(* IEC 61131-3 sources: CodesysTest/export/SX_1195.dev/Plc Logic/Application, 9 files *)

(* ---- AxisData.gvl.st ---- *)
(*#-#-#-#-#-#-#-#-#-#---Declaration---#-#-#-#-#-#-#-#-#-#-#-#-#*)

{attribute 'qualified_only'}
//{attribute 'global_init_slot' := '49994'}
VAR_GLOBAL PERSISTENT

	(* Jaw *)
	jawJogMotionProfile : sctMotionProfile := (
		acceleration := 200,
		deceleration := 200,
		velocity := 2,
		minPosition := 0,
		maxPosition := 5.5,
		current := 30.0
	);
	jawConfig : sctAxisConfig := (
		stepsPerInch := 2410,
		rotationsPerInch := 0.241,
		zeroOffset := 0,
		defaultCurrent := 100.0
	);

	jawOpenMotionProfile : sctMotionProfile := (
		acceleration := 100,
		deceleration := 100,
		velocity := 30.0,
		current := 100.0,
		position := 5.5
	);

	jawCloseMotionProfile : sctMotionProfile := (
		acceleration := 100,
		deceleration := 100,
		velocity := 30.0,
		current := 100.0,
		position := -0.5
	);

	jawPushMotionProfile : sctMotionProfile := (
		acceleration := 100,
		deceleration := 100,
		velocity := 4,
		current := 100.0,
		position := -1
	);

	(* Load Plate *)

	loadPlateConfig : sctAxisConfig := (
		stepsPerInch := 9310,
		rotationsPerInch := 0.931,
		zeroOffset := 0.0
	);

	loadPlateRaiseMotionProfile : sctMotionProfile := (
		acceleration := 300000.0,
		deceleration := 300000.0,
		velocity := 10.0,
		current := 100.0
	);

	loadPlateLowerMotionProfile : sctMotionProfile := (
		acceleration := 300000.0,
		deceleration := 300000.0,
		velocity := 10000.0,
		current := 100.0
	);

	(* IBD *)

	IBDConfig : sctAxisConfig := (
		stepsPerInch := 12500,
		rotationsPerInch := 1.25,
		zeroOffset := 2.0
	);

	IBDJogMotionProfile : sctMotionProfile := (
		acceleration := 0,
		deceleration := 0,
		velocity := 0,
	 	minPosition := 0,
		maxPosition := 0
	);

	IBDOpenMotionProfile : sctMotionProfile := (
		acceleration := 300000.0,
 		deceleration := 300000.0,
		velocity := 10000.0,
		current := 100.0
	);

	IBDCloseMotionProfile : sctMotionProfile := (
		acceleration := 300000.0,
 		deceleration := 300000.0,
		velocity := 10.0,
		current := 50.0
	);

	(* Film Feed *)

	FilmFeedConfig : sctAxisConfig := (
		stepsPerInch := 4900,
		rotationsPerInch := 0.490,
		zeroOffset := 2.0,
		defaultCurrent := 100.0
	);

	FilmFeedJogMotionProfile : sctMotionProfile := (
		acceleration := 200,
		deceleration := 200,
		velocity := 2,
	 	minPosition := -20,
		maxPosition := 20,
		position := 20,
		current := 100
	);

	FilmFeedForwardMotionProfile : sctMotionProfile := (
		acceleration := 75,
 		deceleration := 100,
		velocity := 60,
		position := 17.5,
		current := 100.0
	);

	FilmFeedReverseMotionProfile : sctMotionProfile := (
		acceleration := 50,
 		deceleration := 50,
		velocity := 12,
		position := -1,
		current := 100.0
	);

	FilmFeedPrintMotionProfile : sctMotionProfile := (
		acceleration := 100,
 		deceleration := 100,
		velocity := 12,
		position := -1,
		current := 100.0
	);

	FilmFeedPrintOffsetMotionProfile : sctMotionProfile := (
		acceleration := 75,
 		deceleration := 100,
		velocity := 12,
		position := -1,
		current := 100.0
	);

END_VAR

VAR_GLOBAL
	jaw : sctAxisData := (
		config := jawConfig,
		jogType := eDiscreteMotionType.Absolute
	);

	FilmFeed : sctAxisData := (
		config := FilmFeedConfig,
		jogType := eDiscreteMotionType.Relative
	);

	IBD : sctAxisData := (
		config := IBDConfig,
		jogType := eDiscreteMotionType.Absolute
	);

	loadPlate : sctAxisData := (
		config := loadPlateConfig
	);
END_VAR

(* ---- Counters.gvl.st ---- *)
(*#-#-#-#-#-#-#-#-#-#---Declaration---#-#-#-#-#-#-#-#-#-#-#-#-#*)

{attribute 'qualified_only'}
VAR_GLOBAL
	jawCycleTestCount : FB_MachineCounter(name := 'Jaw Cycle Test Counter');
	baggerCycles : FB_MachineCounter(name := 'Bagger Cycle Counter');
	pressureBarCycles : FB_MachineCounter(name := 'Pressure Bar Cycle Counter');

	(*Counters*)

	//passthroughChanges : FB_MachineCounter(name := 'Passthrough Changes Counter');
	//loadPlateCycles : FB_MachineCounter(name := 'Load Plate Cycle Counter');
	//printerCycles : FB_MachineCounter(name := 'Printer Cycle Counter');
	//motorizedSealFlattenerCycles : FB_MachineCounter(name := 'Motorized Seal Flattener Cycles');
	//bagOpenRetryTotal : FB_MachineCounter(name := 'Bag Open Retry Totals');
END_VAR

(* ---- GlobalData.gvl.st ---- *)
(*#-#-#-#-#-#-#-#-#-#---Declaration---#-#-#-#-#-#-#-#-#-#-#-#-#*)

{attribute 'qualified_only'}
{attribute 'global_init_slot' := '49994'}
VAR_GLOBAL
	SystemLog : FB_InternalLogger;
END_VAR

VAR_GLOBAL CONSTANT
	MAX_LOGGED_ITEMS : UINT := 500;	// Max items to be logged
	STEPS_PER_INCH_IBD : DINT := 1250;
	STEPS_PER_INCH_JAW : DINT := 1250;
	STEPS_PER_INCH_LOAD_PLATE : DINT := 931;
	STEPS_PER_INCH_FILM : DINT := 1000;
	SERIAL_BUFFER_SIZE : BYTE := 50;
	SEAL_TO_PHOTOEYE_DISTANCE : REAL := 3.25;
END_VAR

(* ---- IO.gvl.st ---- *)
(*#-#-#-#-#-#-#-#-#-#---Declaration---#-#-#-#-#-#-#-#-#-#-#-#-#*)

{attribute 'qualified_only'}
{attribute 'global_init_slot' := '50010'}
VAR_GLOBAL
	iptJawNotObstructed : FB_PhysicalDigitalInput(name := 'Jaw Not Obstructed') := (in := iJawNotObstructed);
	iptPrinterDataReady : FB_PhysicalDigitalInput(name := 'Printer Data Ready') := (in := iPrinterDataReady);
	iptPrinterBusy : FB_PhysicalDigitalInput(name := 'Printer Busy') := (in := iPrinterBusy);
	iptBagEdgePhotoeye : FB_PhysicalDigitalInput(name := 'Bag Edge Photoeye') := (in := iBagEdgePhotoeye);
	iptCycleStart : FB_PhysicalDigitalInput(name := 'Cycle Start') := (in := iCycleStart);
	iptPrintHeadLowered : FB_PhysicalDigitalInput(name := 'Printhead Lowered') := (in := iPrintHeadLowered);
	iptJawClosed : FB_PhysicalDigitalInput(name := 'Jaw Closed') := (in := iJawClosed);
	iptJawNearClosed : FB_PhysicalDigitalInput(name := 'Jaw Near Closed') := (in := iJawNearClosed);
	iptBarcodeOK : FB_PhysicalDigitalInput(name := 'Barcode OK') := (in := iBarcodeOK);
	iptBarcodeNG : FB_PhysicalDigitalInput(name := 'Barcode NG') := (in := iBarcodeNG);
	iptLightCurtain : FB_PhysicalDigitalInput(name := 'Light Curtain Clear') := (in := iLightCurtain);
	iptFillerTrigger : FB_PhysicalDigitalInput(name := 'Filler Trigger') := (in := iFillerTrigger);
	iptLHPalmButton : FB_PhysicalDigitalInput(name := 'LH Palm Button') := (in := iLHPalmButton);
	iptRHPalmButton : FB_PhysicalDigitalInput(name := 'RH Palm Button') := (in := iRHPalmButton);
	iptTopCoverClosed : FB_PhysicalDigitalInput(name := 'Top Cover Closed') := (in := iTopCoverClosed);
	iptPrinterRibbonEncoder : FB_PhysicalDigitalInput(name := 'Top Cover Closed') := (in := iPrinterRibbonEncoder);

	outSealWire : FB_PhysicalDigitalOutput(name := 'Seal Wire Output') := (refOutput := oSealWire);
	outLowerPrintHead : FB_PhysicalDigitalOutput(name := 'Lower Printhead') := (refOutput := oLowerPrintHead);
	outRequestPrint : FB_PhysicalDigitalOutput(name := 'Request Print') := (refOutput := oRequestPrint);
	outPrinterRibbonUnwind : FB_PhysicalDigitalOutput(name := 'Ribbon Unwind') := (refOutput := oPrinterRibbonUnwind);
	outTriggerBCV : FB_PhysicalDigitalOutput(name := 'Trigger BCV') := (refOutput := oTriggerBCV);
	outTeachPhotoeye : FB_PhysicalDigitalOutput(name := 'Teach Photoeye') := (refOutput := oTeachPhotoeye);
	outRedStackLight : FB_PhysicalDigitalOutput(name := 'Red Stack Light') := (refOutput := oRedStackLight);
	outGreenStackLight : FB_PhysicalDigitalOutput(name := 'Green Stack Light') := (refOutput := oGreenStackLight);
	outReadyForFiller : FB_PhysicalDigitalOutput(name := 'Ready for Filler') := (refOutput := oReadyForFiller);
	outPalmButton0 : FB_PhysicalDigitalOutput(name := 'Palm Button 0') := (refOutput := oPalmButton0);
	outPalmButton1 : FB_PhysicalDigitalOutput(name := 'Palm Button 1') := (refOutput := oPalmButton1);
END_VAR

(* ---- IO_Mapping.gvl.st ---- *)
(*#-#-#-#-#-#-#-#-#-#---Declaration---#-#-#-#-#-#-#-#-#-#-#-#-#*)

VAR_GLOBAL
	mainIOamax4830Input: ARRAY[0..15] OF universalIOObject;
	mainIOamax4830Output: ARRAY[0..15] OF universalIOObject;
	oSealWire: REFERENCE TO BOOL;
	oLowerPrinthead: Reference to BOOL;
	oRequestPrint: Reference to BOOL;
	oPrinterRibbonUnwind: Reference to BOOL;
	oTriggerBCV: Reference to BOOL;
	oFansEnable: Reference to BOOL;
	oPalmButton0: Reference to BOOL;
	oPalmButton1: Reference to BOOL;
	oPbarClampMotorStart: Reference to BOOL;
	oPbarClampMotorReverse: Reference to BOOL;
	oPbarClampMotorAlarmReset: Reference to BOOL;
	iPrinterServiceRequired: Reference to BOOL;
	iPrinterDataReady: Reference to BOOL;
	iPrinterBusy: Reference to BOOL;
	iBagEdgePhotoeye: Reference to BOOL;
	iCycleStart: Reference to BOOL;
	iPbarClampMotorAlarm: Reference to BOOL;
	iClampHomeSensor: Reference to BOOL;
	iJawNotObstructed: Reference to BOOL;
	iBarcodeOK: Reference to BOOL;
	iBarcodeNG: Reference to BOOL;
	iLightCurtainClear: Reference to BOOL;
	iTopCoverClosed: Reference to BOOL;
	iPrinterRibbonEncoder: REFERENCE TO BOOL;
END_VAR

(* ---- PersistentVars.gvl.st ---- *)
(*#-#-#-#-#-#-#-#-#-#---Declaration---#-#-#-#-#-#-#-#-#-#-#-#-#*)

VAR_GLOBAL RETAIN PERSISTENT
	// Generated instance path of persistent variable
	PLC_PRG_1.baggerCM.dualMotorPassthrough.factoryHomeJaw: BOOL;
	// Generated instance path of persistent variable
	HMIData.bagsMade: UDINT;
	// Generated instance path of persistent variable
	HMIData.batchEnable: BOOL;
	// Generated instance path of persistent variable
	HMIData.batchSetting: UDINT := UDINT#10;
	// Generated instance path of persistent variable
	HMIData.batchCount: UDINT;
	// Generated instance path of persistent variable
	HMIData.headCycleCount: UDINT;
	// Generated instance path of persistent variable
	HMIData.pressureBarOpenDelay: REAL;
	// Generated instance path of persistent variable
	HMIData.pressureBarCloseDelay: REAL;
	// Generated instance path of persistent variable
	HMIData.passthroughSetting: REAL := REAL#5.5;
	// Generated instance path of persistent variable
	HMIData.sealBarDwell: REAL := REAL#0.2;
	// Generated instance path of persistent variable
	HMIData.sealBarCool: REAL := REAL#0.4;
	// Generated instance path of persistent variable
	HMIData.bagSkirtLength: REAL := 2.0;
	// Generated instance path of persistent variable
	HMIData.bagLength: REAL := REAL#17.62;
	// Generated instance path of persistent variable
	HMIData.bagWidth: REAL := 11.0;
	// Generated instance path of persistent variable
	HMIData.bagThickness: REAL := REAL#2.5;
	// Generated instance path of persistent variable
	HMIData.bagForwardSpeed: UDINT := UDINT#40;
	// Generated instance path of persistent variable
	HMIData.bagReverseSpeed: UDINT := UDINT#8;
	// Generated instance path of persistent variable
	HMIData.printSpeed: UINT := UINT#6;
	// Generated instance path of persistent variable
	HMIData.printLength: REAL := REAL#1.25;
	// Generated instance path of persistent variable
	HMIData.printOffset: REAL := REAL#9;
	// Generated instance path of persistent variable
	HMIData.fillerCountSetting: UDINT;
	// Generated instance path of persistent variable
	HMIData.fillerCurrentCount: UDINT;
	// Generated instance path of persistent variable
	HMIData.fillerDropTime: REAL;
	// Generated instance path of persistent variable
	HMIData.loadPlateDelay: REAL;
	// Generated instance path of persistent variable
	HMIData.loadPlateDwell: REAL := REAL#0.1;
	// Generated instance path of persistent variable
	HMIData.IBDInUse: BOOL;
	// Generated instance path of persistent variable
	HMIData.IBDInstalled: BOOL := FALSE;
	// Generated instance path of persistent variable
	HMIData.jawCloseDelay: REAL := REAL#0.1;
	// Generated instance path of persistent variable
	HMIData.jawClosePositionSetting: REAL := REAL#-0.45;
	// Generated instance path of persistent variable
	HMIData.lastCycleTime: REAL;
	// Generated instance path of persistent variable
	HMIData.bagDropClearanceDwell: REAL := REAL#0.5;
	// Generated instance path of persistent variable
	HMIData.averageCycleTime: REAL;
	// Generated instance path of persistent variable
	HMIData.currentJobID: INT;
	// Generated instance path of persistent variable
	HMIData.separateBeforeSeal: BOOL := TRUE;
	// Generated instance path of persistent variable
	HMIData.partsCounterEnable: BOOL;
	// Generated instance path of persistent variable
	HMIData.partsCounterCount: UDINT;
	// Generated instance path of persistent variable
	HMIData.partsCounterSetting: UDINT;
	// Generated instance path of persistent variable
	HMIData.consecutiveBagsEnable: BOOL;
	// Generated instance path of persistent variable
	HMIData.consecutiveBagsCount: UDINT;
	// Generated instance path of persistent variable
	HMIData.consecutiveBagsSetting: UDINT;
	// Generated instance path of persistent variable
	HMIData.printerInstalled: BOOL := FALSE;
	// Generated instance path of persistent variable
	HMIData.printerInUse: BOOL := FALSE;
	// Generated instance path of persistent variable
	HMIData.printerCancelRequest: BOOL;
	// Generated instance path of persistent variable
	HMIData.barcodeVerifierInstalled: BOOL := FALSE;
	// Generated instance path of persistent variable
	HMIData.barcodeGoodReadCount: UDINT;
	// Generated instance path of persistent variable
	HMIData.barcodeBadReadCount: UDINT;
	// Generated instance path of persistent variable
	HMIData.barcodeBadReadFaultSetting: UDINT := UDINT#1;
	// Generated instance path of persistent variable
	HMIData.barcodeStartPosition: REAL := REAL#4.5;
	// Generated instance path of persistent variable
	HMIData.barcodeScanDistance: REAL := REAL#0.1;
	// Generated instance path of persistent variable
	HMIData.barcodeVerifierInUse: BOOL;
	// Generated instance path of persistent variable
	HMIData.loadPlateInstalled: BOOL := FALSE;
	// Generated instance path of persistent variable
	HMIData.loadPlateLoweredPositionSetting: REAL := 0.0;
	// Generated instance path of persistent variable
	HMIData.loadPlateRaisedPositionSetting: REAL := 1.0;
	// Generated instance path of persistent variable
	HMIData.loadPlateInUse: BOOL;
	// Generated instance path of persistent variable
	HMIData.fillerEnable: BOOL;
	// Generated instance path of persistent variable
	HMIData.autoModeEnable: BOOL;
	// Generated instance path of persistent variable
	HMIData.autoModeDwell: REAL;
	// Generated instance path of persistent variable
	HMIData.dryCycleEnable: BOOL;
	// Generated instance path of persistent variable
	HMIData.standbyTimeSetting: REAL := REAL#5;
	// Generated instance path of persistent variable
	HMIData.jawClampTime: REAL := REAL#1;
	// Generated instance path of persistent variable
	HMIData.jawClampReverseTime: REAL := REAL#1;
	// Generated instance path of persistent variable
	HMIData.jawClampInterval: REAL := REAL#2;
	// Generated instance path of persistent variable
	HMIData.jawEnableClamping: BOOL;
	// Generated instance path of persistent variable
	HMIData.jawCycleTestCycles: DINT;
	// Generated instance path of persistent variable
	HMIData.jawClampTestCycles: DINT;
	// Generated instance path of persistent variable
	HMIData.filmFeedTestCycles: DINT;
	// Generated instance path of persistent variable
	HMIData.jawEnableMotion: BOOL;
	// Generated instance path of persistent variable
	HMIData.filmEnableMotion: BOOL;
	// Generated instance path of persistent variable
	HMIData.printer300DPI: BOOL;
	// Generated instance path of persistent variable
	AxisData.jawJogMotionProfile: sctMotionProfile := STRUCT(acceleration := 200.0, deceleration := 200.0, velocity := 2.0, minPosition := REAL#0.0, maxPosition := 5.5, current := REAL#30);
	// Generated instance path of persistent variable
	AxisData.jawConfig: sctAxisConfig := STRUCT(stepsPerInch := 2410.0, rotationsPerInch := REAL#0.241, zeroOffset := 0.0, defaultCurrent := REAL#100);
	// Generated instance path of persistent variable
	AxisData.jawOpenMotionProfile: sctMotionProfile := STRUCT(acceleration := 100.0, deceleration := 100.0, velocity := REAL#30, current := REAL#100, position := REAL#5.5);
	// Generated instance path of persistent variable
	AxisData.jawCloseMotionProfile: sctMotionProfile := STRUCT(acceleration := 100.0, deceleration := 100.0, velocity := REAL#30, current := REAL#100, position := REAL#-0.5);
	// Generated instance path of persistent variable
	AxisData.jawPushMotionProfile: sctMotionProfile := STRUCT(acceleration := 100.0, deceleration := 100.0, velocity := 4.0, current := REAL#100, position := -1.0);
	// Generated instance path of persistent variable
	AxisData.loadPlateConfig: sctAxisConfig := STRUCT(stepsPerInch := 9310.0, rotationsPerInch := REAL#0.931, zeroOffset := REAL#0);
	// Generated instance path of persistent variable
	AxisData.loadPlateRaiseMotionProfile: sctMotionProfile := STRUCT(acceleration := REAL#300000, deceleration := REAL#300000, velocity := REAL#10, current := REAL#100);
	// Generated instance path of persistent variable
	AxisData.loadPlateLowerMotionProfile: sctMotionProfile := STRUCT(acceleration := REAL#300000, deceleration := REAL#300000, velocity := REAL#10000, current := REAL#100);
	// Generated instance path of persistent variable
	AxisData.IBDConfig: sctAxisConfig := STRUCT(stepsPerInch := 12500.0, rotationsPerInch := REAL#1.25, zeroOffset := REAL#2);
	// Generated instance path of persistent variable
	AxisData.IBDJogMotionProfile: sctMotionProfile := STRUCT(acceleration := 0.0, deceleration := 0.0, velocity := 0.0, minPosition := 0.0, maxPosition := 0.0);
	// Generated instance path of persistent variable
	AxisData.IBDOpenMotionProfile: sctMotionProfile := STRUCT(acceleration := REAL#300000, deceleration := REAL#300000, velocity := REAL#10000, current := REAL#100);
	// Generated instance path of persistent variable
	AxisData.IBDCloseMotionProfile: sctMotionProfile := STRUCT(acceleration := REAL#300000, deceleration := REAL#300000, velocity := REAL#10, current := REAL#50);
	// Generated instance path of persistent variable
	AxisData.FilmFeedConfig: sctAxisConfig := STRUCT(stepsPerInch := 4900.0, rotationsPerInch := REAL#0.49, zeroOffset := REAL#2, defaultCurrent := REAL#100);
	// Generated instance path of persistent variable
	AxisData.FilmFeedJogMotionProfile: sctMotionProfile := STRUCT(acceleration := 10.0, deceleration := 200.0, velocity := 100.0, minPosition := -20.0, maxPosition := 20.0, position := 20.0, current := 100.0);
	// Generated instance path of persistent variable
	AxisData.FilmFeedForwardMotionProfile: sctMotionProfile := STRUCT(acceleration := 75.0, deceleration := 100.0, velocity := 60.0, position := REAL#17.5, current := REAL#100);
	// Generated instance path of persistent variable
	AxisData.FilmFeedReverseMotionProfile: sctMotionProfile := STRUCT(acceleration := 50.0, deceleration := 50.0, velocity := 12.0, position := -1.0, current := REAL#100);
	// Generated instance path of persistent variable
	AxisData.FilmFeedPrintMotionProfile: sctMotionProfile := STRUCT(acceleration := 100.0, deceleration := 100.0, velocity := 12.0, position := -1.0, current := REAL#100);
	// Generated instance path of persistent variable
	AxisData.FilmFeedPrintOffsetMotionProfile: sctMotionProfile := STRUCT(acceleration := 75.0, deceleration := 100.0, velocity := 12.0, position := -1.0, current := REAL#100);
END_VAR

(* ---- IO_Map.pou.st ---- *)
(*#-#-#-#-#-#-#-#-#-#---Declaration---#-#-#-#-#-#-#-#-#-#-#-#-#*)

PROGRAM IO_Map
VAR
END_VAR
(*#-#-#-#-#-#-#-#-#-#---Implementation---#-#-#-#-#-#-#-#-#-#-#-#-#*)

//Output Configuration

oSealWire REF= IO_Mapping.mainIOamax4830Output[0].discreteSignal;
oLowerPrinthead REF= IO_Mapping.mainIOamax4830Output[1].discreteSignal;
oRequestPrint REF=IO_Mapping.mainIOamax4830Output[2].discreteSignal;
oPrinterRibbonUnwind REF=IO_Mapping.mainIOamax4830Output[3].discreteSignal;
oTriggerBCV REF=IO_Mapping.mainIOamax4830Output[4].discreteSignal;
//IO_Mapping.mainIOamax4830Output[5].discreteSignal;
oFansEnable REF=IO_Mapping.mainIOamax4830Output[6].discreteSignal;
//IO_Mapping.mainIOamax4830Output[7].discreteSignal;
//IO_Mapping.mainIOamax4830Output[8].discreteSignal;
oPalmButton0 REF=IO_Mapping.mainIOamax4830Output[9].discreteSignal;
oPalmButton1 REF=IO_Mapping.mainIOamax4830Output[10].discreteSignal;
oPbarClampMotorStart REF=IO_Mapping.mainIOamax4830Output[11].discreteSignal;
oPbarClampMotorReverse REF=IO_Mapping.mainIOamax4830Output[12].discreteSignal;
oPbarClampMotorAlarmReset REF=IO_Mapping.mainIOamax4830Output[13].discreteSignal;
//IO_Mapping.mainIOamax4830Output[14].discreteSignal;
//IO_Mapping.mainIOamax4830Output[15].discreteSignal;

IO_Mapping.mainIOamax4830Output[0].signalCommonName := 'O0\0: Seal Wire';
IO_Mapping.mainIOamax4830Output[1].signalCommonName := 'O0\1: Lower Print Head';
IO_Mapping.mainIOamax4830Output[2].signalCommonName := 'O0\2: Request Print';
IO_Mapping.mainIOamax4830Output[3].signalCommonName := 'O0\3: Printer Ribbon Unwind';
IO_Mapping.mainIOamax4830Output[4].signalCommonName := 'O0\4: Trigger Barcode Verification';
IO_Mapping.mainIOamax4830Output[5].signalCommonName := 'O0\5: Spare';
IO_Mapping.mainIOamax4830Output[6].signalCommonName := 'O0\6: Fans Enable';
IO_Mapping.mainIOamax4830Output[7].signalCommonName := 'O0\7: Spare';
IO_Mapping.mainIOamax4830Output[8].signalCommonName := 'O0\8: Spare';
IO_Mapping.mainIOamax4830Output[9].signalCommonName := 'O0\9: Palm Button 0';
IO_Mapping.mainIOamax4830Output[10].signalCommonName := 'O0\10: Palm Button 1';
IO_Mapping.mainIOamax4830Output[11].signalCommonName := 'O0\11: Pbar Clamp Motor Start';
IO_Mapping.mainIOamax4830Output[12].signalCommonName := 'O0\12: Pbar Clamp Motor Reverse';
IO_Mapping.mainIOamax4830Output[13].signalCommonName := 'O0\13: Pbar Clamp Motor Alarm Reset';
IO_Mapping.mainIOamax4830Output[14].signalCommonName := 'O0\14: Spare';
IO_Mapping.mainIOamax4830Output[15].signalCommonName := 'O0\15: Spare';

//Input Configuration

iPrinterServiceRequired REF= IO_Mapping.mainIOamax4830Input[0].discreteSignal;
iPrinterDataReady REF= IO_Mapping.mainIOamax4830Input[1].discreteSignal;
iPrinterBusy REF= IO_Mapping.mainIOamax4830Input[2].discreteSignal;
iBagEdgePhotoeye REF= IO_Mapping.mainIOamax4830Input[3].discreteSignal;
iCycleStart REF= IO_Mapping.mainIOamax4830Input[4].discreteSignal;
iPbarClampMotorAlarm REF= IO_Mapping.mainIOamax4830Input[5].discreteSignal;
iClampHomeSensor REF= IO_Mapping.mainIOamax4830Input[6].discreteSignal;
iJawNotObstructed REF= IO_Mapping.mainIOamax4830Input[7].discreteSignal;
iBarcodeOK REF= IO_Mapping.mainIOamax4830Input[8].discreteSignal;
iBarcodeNG REF= IO_Mapping.mainIOamax4830Input[9].discreteSignal;
iLightCurtainClear REF= IO_Mapping.mainIOamax4830Input[10].discreteSignal;
//IO_Mapping.mainIOamax4830Input[11].discreteSignal;
//IO_Mapping.mainIOamax4830Input[12].discreteSignal;
//IO_Mapping.mainIOamax4830Input[13].discreteSignal;
iTopCoverClosed REF= IO_Mapping.mainIOamax4830Input[14].discreteSignal;
iPrinterRibbonEncoder REF= IO_Mapping.mainIOamax4830Input[15].discreteSignal;

IO_Mapping.mainIOamax4830Input[0].signalCommonName := 'I0\0: Printer Service Required';
IO_Mapping.mainIOamax4830Input[1].signalCommonName := 'I0\1: Printer Data Ready';
IO_Mapping.mainIOamax4830Input[2].signalCommonName := 'I0\2: Printer Busy';
IO_Mapping.mainIOamax4830Input[3].signalCommonName := 'I0\3: Bag Edge Detect Photoeye';
IO_Mapping.mainIOamax4830Input[4].signalCommonName := 'I0\4: Cycle Start';
IO_Mapping.mainIOamax4830Input[5].signalCommonName := 'I0\5: Pbar Clamp Motor Alarm';
IO_Mapping.mainIOamax4830Input[6].signalCommonName := 'I0\6: Clamp Home Sensor';
IO_Mapping.mainIOamax4830Input[7].signalCommonName := 'I0\7: Jaw Not Obstructed';
IO_Mapping.mainIOamax4830Input[8].signalCommonName := 'I0\8: Bracode OK';
IO_Mapping.mainIOamax4830Input[9].signalCommonName := 'I0\9: Bracode NG';
IO_Mapping.mainIOamax4830Input[10].signalCommonName := 'I0\10: Light Curtain Clear';
IO_Mapping.mainIOamax4830Input[11].signalCommonName := 'I0\11: Spare';
IO_Mapping.mainIOamax4830Input[12].signalCommonName := 'I0\12: Spare';
IO_Mapping.mainIOamax4830Input[13].signalCommonName := 'I0\13: Spare';
IO_Mapping.mainIOamax4830Input[14].signalCommonName := 'I0\14: Top Cover Closed';
IO_Mapping.mainIOamax4830Input[15].signalCommonName := 'I0\15: Printer Ribbon Encoder';

(* ---- PLC_PRG.pou.st ---- *)
(*#-#-#-#-#-#-#-#-#-#---Declaration---#-#-#-#-#-#-#-#-#-#-#-#-#*)

PROGRAM PLC_PRG
VAR
	firstScanDone: BOOL;
	cycleStartONS : FB_ONS;
	powerUpFrontJawMotor : MC_Power;
	powerUpRearJawMotor : MC_Power;
	powerUpBothJawMotors : MC_Power;
	powerUpLoadPlateMotor : MC_Power;
	powerUpBagDeliveryMotor : MC_Power;
	powerUpIBDMotor : MC_Power;
	UN00_SXMachine : FB_UN00_SharpMachine(name := 'UN00 - Sharp SX');
	EM01_SXBaggerHead : EM01_BaggerHead(name := 'EM01 - SX Bagger Head');
	EM02_SXDischarge : EM02_Discharge(name := 'EM02 - SX Discharge');
	baggerCM : EM01_Bagger_Control_Modules;
	bannerManager : FB_BannerManager;
	palmButton : FB_BannerPalmButton;
	topCoverLiftedFault : FB_Fault(name := 'Top Cover Lifeted During Cycle');
	amazonBPM : FB_AmazonThroughput();
	printerLabel : FB_PrinterSerial();
	autoModeTimer : Standard.TON;
	autoModeKeepCycling : BOOL;
	autoModeInitiateCycleONS : FB_ONS;
	cycleComplete : FB_ONS;
	hIecTask : RTS_IEC_HANDLE;//Declaration of the variable hIecTask
	teachPhotoeyeTimer : Standard.TOF() := (PT := T#3S);
	standbyTimer : Standard.TON;
END_VAR(*#-#-#-#-#-#-#-#-#-#---Implementation---#-#-#-#-#-#-#-#-#-#-#-#-#*)

//	Program: PLC_PRG
//	Description: Base program for the 1179/1181 SX.
//		Control modules are set up in EM01_Bagger_Control_Modules
//		Automatic cycle control is set up in POUs - EM01_BaggerHead_Automode.Executing
// 		This program sets up machine specific contol modules and interfaces to the HMI.
//
//	Created by: Ben Hess
//	Created Date:
(*

PackML Machine States for Sharp Baggers

+---------------------------------------------------------------------------------------+
| +----------------+          +----------------+         +----------------+             |
| |                |          |                |         |                |             |
| |      Idle      |--------->|    Starting    |-------->|     Execute    |             |
| |                |          |                |         |                |             |
| +----------------+          +----------------+         +----------------+             |
|          ^                                                                            |
|          |                                                                            |
|          |                                                                            |
|          |                                                                            |
| +----------------+                                                                    |
| |                |                                                                    |
| |   Resetting    |                                                                    |
| |                |                                                                    |
| +----------------+                                                                    |
|          ^                                                                            |
+---------------------------------------------------------------------------------------+
|          |                     |                                                      |
|          |                     |                                                      |
+---------------------------------------------------------------------------------------+
|          |                     v          |                                   |
| +----------------+    +----------------+  |                                   |
| |                |    |                |  |                                   |
| |    Stopped     |<-- |    Stopping    |  |                                   v
| |                |    |                |  |    +----------------+    +----------------+
| +----------------+    +----------------+  |    |                |    |                |
|                                ^          |    |    Aborted     | <- |    Aborting    |
|                                |          |    |                |    |                |
|                       +----------------+  |    +----------------+    +----------------+
|                       |                |  |             |
|                       |    Clearing    |  |             |
|                       |                |<---------------|
|                       +----------------+  |
+-------------------------------------------+
*)

// Initialze global objects on first scan
IF NOT firstScanDone THEN
	GlobalObjects.CollectionOfInitialzable.InitializeAll();
	GlobalObjects.CollectionOfLoggable.RegisterAll(internalLogger := Globals.SystemLog);
	GlobalObjects.CollectionOfFaults.FaultUpdateForHMI();
	hIecTask := IecTaskGetCurrent(0);
	IecTaskDisableWatchdog(hIecTask); // Watchdog disabled
END_IF

// Use fault collection for faultActive indication
HMIData.faultActive := GlobalObjects.CollectionOfActiveFaults.faultActive;

(* Cycle start conditions *)
// Auto mode dwell timer
autoModeTimer(PT := TO_TIME(HMIData.autoModeDwell * 1000), IN := autoModeKeepCycling AND UN00_SXMachine.currentState = PACK_ML.State.Execute AND NOT HMIData.inCycle);
// Start from Cycle Start input
cycleStartONS(clk := iCycleStart);
// All start conditions
IF HMIData.initiateCycle OR cycleStartONS.OSR OR autoModeTimer.Q THEN
	IF UN00_SXMachine.currentState = PACK_ML.State.Execute AND NOT HMIData.inCycle THEN
		EM01_SXBaggerHead.StartCycle();
		IF HMIData.autoModeEnable THEN
			autoModeKeepCycling := TRUE;
		END_IF
	END_IF
	HMIData.initiateCycle := FALSE;
END_IF
// Unlatch flag for auto mode when faulted or stopped
IF UN00_SXMachine.currentState <> PACK_ML.State.Execute OR HMIData.ackAllFaults OR NOT HMIData.autoModeEnable THEN
	autoModeKeepCycling := FALSE;
END_IF

// Fault FB's execute automatically to handle acking and clearing without having to be run in each FB that contains them
IF firstScanDone THEN
	GlobalObjects.CollectionOfExecutable.ExecuteAll();
END_IF

// Power up all motors
powerUpFrontJawMotor(Enable := TRUE, Axis := baggerCM.jawFrontMotor);
powerUpFrontJawMotor.DriveStart := TRUE;
powerUpFrontJawMotor.RegulatorOn := TRUE;

powerUpRearJawMotor(Enable := TRUE, Axis := baggerCM.jawRearMotor);
powerUpRearJawMotor.DriveStart := TRUE;
powerUpRearJawMotor.RegulatorOn := TRUE;

powerUpBothJawMotors(Enable := TRUE, Axis := baggerCM.jawBothMotors);
powerUpBothJawMotors.DriveStart := TRUE;
powerUpBothJawMotors.RegulatorOn := TRUE;

powerUpLoadPlateMotor(Enable := HMIData.loadPlateInstalled, Axis := baggerCM.loadPlateMotor);
powerUpLoadPlateMotor.DriveStart := HMIData.loadPlateInstalled;
powerUpLoadPlateMotor.RegulatorOn := HMIData.loadPlateInstalled;

powerUpBagDeliveryMotor(Enable := TRUE, Axis := baggerCM.bagDeliveryFrontMotor);
powerUpBagDeliveryMotor.DriveStart := TRUE;
powerUpBagDeliveryMotor.RegulatorOn := TRUE;

powerUpIBDMotor(Enable := HMIData.IBDInstalled, Axis := baggerCM.IBDMotor);
powerUpIBDMotor.DriveStart := HMIData.IBDInstalled;
powerUpIBDMotor.RegulatorOn := HMIData.IBDInstalled;

// Disable Modbus device tree objects if option not installed
IF NOT HMIData.loadPlateInstalled THEN
	Load_Plate_Motor.Enable := FALSE;
ELSE
	Load_Plate_Motor.Enable := TRUE;
END_IF

IF NOT HMIData.IBDInstalled THEN
	IBD_Motor.Enable := FALSE;
ELSE
	IBD_Motor.Enable := TRUE;
END_IF

// Barcode Verifier manual trigger
IF HMIData.barcodeVerifierTrigger THEN
	baggerCM.barcodeVerifier.TriggerImmediate();
	HMIData.barcodeVerifierTrigger := FALSE;
END_IF

// Printer sample label sending
IF HMIData.sendSampleLabels AND NOT printerLabel.xExecute THEN
	printerLabel.xExecute := TRUE;
	printerLabel.sendSampleLabel := TRUE;
	printerLabel.sendClearLabel := FALSE;
	HMIData.sendSampleLabels := FALSE;
ELSIF HMIData.clearAllLabels AND NOT printerLabel.xExecute THEN
	printerLabel.xExecute := TRUE;
	printerLabel.sendSampleLabel := FALSE;
	printerLabel.sendClearLabel := TRUE;
	HMIData.clearAllLabels := FALSE;
END_IF

IF printerLabel.xDone THEN
	printerLabel.xExecute := FALSE;
END_IF
printerLabel();

// Run collection of bagger control modules
baggerCM();

// Set bagger head control modules and run head Equipment Module
EM01_SXBaggerHead(
	bagOpenFingers:= baggerCM.dummyBOF,
	sealFlatteners:= baggerCM.dummySealFlatteners,
	sealer:= baggerCM.sealWire,
	pressureBar:= baggerCM.dualMotorPassthrough,
	printer:= baggerCM.labelPrinter,
	bagDelivery:= baggercm.bagDelivery,
	vacuumBagOpen:= baggerCM.dummyVacuumCups,
	IBD:= baggerCM.IBD,
	loadPlate:= baggerCM.loadPlate,
	barcodeVerifier:= baggerCM.barcodeVerifier,
	bagOpenAssistEnabled:= FALSE,
	bagOpenSensorEnabled:= FALSE,
	cancelPrint := HMIData.printerCancelRequest,
	separateBeforeSealEnabled:= HMIData.separateBeforeSeal,
	bagOpenRetrySetting:= ,
	newJobLoaded:= ,
	vacuumDwell:= ,
	bagOpenRetryCount=> ,
	failedToOpenBag=> );

// Run discharge Equipment Module
EM02_SXDischarge();

// Machine unit
UN00_SXMachine(faultActive:= HMIData.faultActive, resetMachine := HMIData.ackAllFaults, homeMachine := HMIData.homeMachine, currentState=> , baggerHead:= EM01_SXBaggerHead, discharge:= EM02_SXDischarge);

// Trigger fault if top cover lifted during cycle
IF HMIData.inCycle AND NOT iTopCoverClosed THEN
	topCoverLiftedFault.Trigger();
END_IF

// Banner palm button has 4 states - off, solid green, 50/50 green/white rotating, and flashing red
palmButton(
	baggerReady:= UN00_SXMachine.currentState = PACK_ML.State.Execute,
	baggerFaulted:= HMIData.faultActive,
	baggerInCycle:= HMIData.inCycle,
	palmState0Output=> oPalmButton0,
	palmState1Output=> oPalmButton1);

// Standby timer - timeout and turn off fans if not cycled. Turn them back on once reset
standbyTimer(IN := NOT HMIData.inCycle AND UN00_SXMachine.currentState = PACK_ML.State.Execute, PT := TO_TIME(HMIData.standbyTimeSetting * 60 * 1000));
IF standbyTimer.Q AND HMIData.standbyTimeSetting > 0 THEN
	UN00_SXMachine.StopMachine();
	HMIData.standbyActive := TRUE;
END_IF

IF HMIData.ackAllFaults THEN
	HMIData.standbyActive := FALSE;
END_IF

oFansEnable := NOT HMIData.standbyActive;

//
// HMI Mapping
//

// Send the list of active fault strings to HMI for viewing
HMIData.activeFaults := GlobalObjects.CollectionOfActiveFaults.ObjNames;

// In cycle indication
HMIData.inCycle := UN00_SXMachine.baggerManager.BaggerAutoMode.baggerCycleActive;

// PackML state to string for HMI
HMIData.currentPackMLState := UN00_SXMachine.baggerManager.BaggerAutoMode.currentBaggerState;

// Banner manager takes care of the Multistate lamp used as a banner on the proface
bannerManager(
	baggerNotReady:= NOT (UN00_SXMachine.currentState = PACK_ML.State.Execute) AND NOT HMIData.standbyActive,
	baggerReady:= UN00_SXMachine.currentState = PACK_ML.State.Execute AND NOT HMIData.inCycle AND NOT HMIData.standbyActive,
	baggerInCycle:= HMIData.inCycle,
	noBagCoveringEye:= baggerCM.bagDelivery.noBagOverEye.Active,
	bagFailedToSeperate:= baggerCM.bagDelivery.bagFailedToSeparate.Active,
	pbarObstruction:= baggerCM.dualMotorPassthrough.pressureBarObstructed.Active,
	lightCurtainViolation:= ,
	printHeadFTR:= baggerCM.labelPrinter.printHeadFailToRaise.Active,
	printHeadFTL:= baggerCM.labelPrinter.printHeadFailToLower.Active,
	barcodeFault:= EM01_SXBaggerHead.barcodeVerificationFailed.Active,
	tooManyPartsCounted:= ,
	jawFailedToClose:= baggerCM.dualMotorPassthrough.failedToClose.Active,
	jawFailedToHome:= baggerCM.dualMotorPassthrough.failedToHome.Active,
	filmFeedMotorFault:= baggerCM.bagDelivery.motorFault.Active,
	filmFeedMotorCommF:= baggerCM.bagDelivery.motorCommFault.Active,
	jawMotionFault:= baggerCM.dualMotorPassthrough.bothMotorsFault.Active,
	waitingOnPrinter:= UN00_SXMachine.baggerManager.BaggerAutoMode.releaseAndFeedSubState = RELEASE_FEED_STATES.WaitForPrinter,
	waitingOnFiller:= ,
	batchCounterDone:= ,
	jawNotHomed:= NOT baggerCM.dualMotorPassthrough.IsHomed AND NOT HMIData.inCycle,
	cycleBaggerTForFiller:= ,
	machineNotTested:=  HMIData.bagsMade < 1000,
	loadPlateMotorNotHomed:= NOT baggerCM.loadPlate.IsHomed AND baggerCM.loadPlate.OptionActive,
	loadPlateMotorFaulted:= baggerCM.loadPlate.motorFault.Active,
	loadPlateMotorCommF:= baggerCM.loadPlate.motorCommFault.Active,
	topCoverLiftedFault:= topCoverLiftedFault.Active,
	topCoverLiftedWarning:= NOT iTopCoverClosed AND NOT HMIData.inCycle,
	IBDMotorNotHomed:= NOT baggerCM.IBD.IsHomed AND baggerCM.IBD.OptionActive AND NOT HMIData.inCycle,
	IBDMotorFaulted:= baggerCM.IBD.IBDMotorFault.Active,
	IBDMotorCommF:= baggerCM.IBD.IBDMotorCommFault.Active,
	printerRibbonFault := baggerCM.labelPrinter.ribbonFault.Active,
	printerServiceRequired := baggerCM.labelPrinter.serviceRequired.Active,
	jawFailedToOpen:= baggerCM.dualMotorPassthrough.failedToOpen.Active,
	IBDFailedToClose:= ,
	IBDFailedToOpen:= baggerCM.IBD.failedToOpen.Active,
	baggerInStandby := HMIData.standbyActive,
	messageDisplayIndication=> HMIData.bannerMessageIndication);

// Ready indications for bagger control modules
HMIData.printerReady := baggerCM.labelPrinter.Ready;
HMIData.bagDeliveryReady := baggerCM.bagDelivery.Ready;
HMIData.loadPlateReady := baggerCM.loadPlate.Ready;
HMIData.jawReady := baggerCM.dualMotorPassthrough.Ready;
HMIData.bcvReady := baggerCM.barcodeVerifier.Ready;
HMIData.IBDReady := baggerCM.IBD.Ready;

// Motor data to HMI for troubleshooting
HMIData.frontJawMotorData.ActPos := baggerCM.jawFrontMotor.ActPos;
HMIData.frontJawMotorData.CommandedPos := baggerCM.jawFrontMotor.TargetPosDist;
HMIData.frontJawMotorData.CurrentAlarmCode := baggerCM.jawFrontMotor.alarmCode;

HMIData.rearJawMotorData.ActPos := baggerCM.jawRearMotor.ActPos;
HMIData.rearJawMotorData.CommandedPos := baggerCM.jawRearMotor.TargetPosDist;
HMIData.rearJawMotorData.CurrentAlarmCode := baggerCM.jawRearMotor.alarmCode;

HMIData.IBDMotorData.ActPos := baggerCM.IBDMotor.ActPos;
HMIData.IBDMotorData.CommandedPos := baggerCM.IBDMotor.TargetPosDist;
HMIData.IBDMotorData.CurrentAlarmCode := baggerCM.IBDMotor.alarmCode;

HMIData.loadPlateMotorData.ActPos := baggerCM.loadPlateMotor.ActPos;
HMIData.loadPlateMotorData.CommandedPos := baggerCM.loadPlateMotor.TargetPosDist;
HMIData.loadPlateMotorData.CurrentAlarmCode := baggerCM.loadPlateMotor.alarmCode;

HMIData.bagDeliveryMotorData.alarmCode := baggerCM.bagDeliveryFrontMotor.alarmCode;
HMIData.bagDeliveryMotorData.statusCode := baggerCM.bagDeliveryFrontMotor.statusCode;

// Cycle time and bags made counters
HMIData.cycleTime := UN00_SXMachine.baggerManager.BaggerAutoMode.cycleTime;
HMIData.inCycle := UN00_SXMachine.baggerManager.BaggerAutoMode.cycleTimer.IN;
cycleComplete(CLK := UN00_SXMachine.baggerManager.BaggerAutoMode.cycleComplete);
IF cycleComplete.OSR THEN
	HMIData.bagsMade := HMIData.bagsMade + 1;
END_IF

// Printer and Barcode Verifier combination enable/disable
HMIData.printerAndVerifierEnableIndication := HMIData.printerInUse AND HMIData.barcodeVerifierInUse;
IF HMIData.printerAndVerifierEnablePB THEN
	IF HMIData.printerAndVerifierEnableIndication THEN
		HMIData.printerInUse := FALSE;
		HMIData.barcodeVerifierInUse := FALSE;
	ELSE
		HMIData.printerInstalled := TRUE;
		HMIData.barcodeVerifierInstalled := TRUE;
		HMIData.printerInUse := TRUE;
		HMIData.barcodeVerifierInUse := TRUE;
	END_IF
	HMIData.printerAndVerifierEnablePB := FALSE;
END_IF

// Position Indications for service commands
HMIData.jawService.extendedFeedback := baggerCM.dualMotorPassthrough.IsFullyOpen;
HMIData.jawService.retractedFeedback := baggerCM.dualMotorPassthrough.IsFullyClosed;

HMIData.IBDService.extendedFeedback := baggerCM.IBD._isFullyOpen;
HMIData.IBDService.retractedFeedback := NOT baggerCM.IBD._isFullyOpen;

// HMIData.printHeadService.extendedFeedback := iPrintHeadLowered;
// HMIData.printHeadService.retractedFeedback := NOT iPrintHeadLowered;

// Amazon Bags per minute throughput calculator
amazonBPM(
	inCycle:= HMIData.inCycle,
	runtimeTimeout:= ,
	reset:= HMIData.BPMReset,
	BPM=> HMIData.BPMBagsPerMinute,
	BPMCycles=> HMIData.BPMBagsMade,
	BPMSeconds=> ,
	BPMIndication=> HMIData.BPMActiveTime);

// Set first scan complete flag
firstScanDone := TRUE;

(* ---- PLC_PRG_1.pou.st ---- *)
(*#-#-#-#-#-#-#-#-#-#---Declaration---#-#-#-#-#-#-#-#-#-#-#-#-#*)

PROGRAM PLC_PRG_1
VAR
	firstScanDone: BOOL;
	firstAborted :BOOL:=TRUE;
	cycleStartONS : FB_ONS;
	powerUpFrontJawMotor : MC_Power;
	powerUpRearJawMotor : MC_Power;
	powerUpBothJawMotors : MC_Power;
	powerUpLoadPlateMotor : MC_Power;
	powerUpBagDeliveryMotor : MC_Power;
	powerUpIBDMotor : MC_Power;
	UN00_SXMachine : FB_UN00_SharpMachine(name := 'UN00 - Sharp SX');
	EM01_SXBaggerHead : EM01_BaggerHead(name := 'EM01 - SX Bagger Head');
	EM02_SXDischarge : EM02_Discharge(name := 'EM02 - SX Discharge');
	baggerCM : EM01_BaggerCM;
	dischargeCM : EM02_DischargeCM;
	bannerManager : FB_BannerManager;
	hmiFaultMessage : FB_FaultMessageHandler;
	palmButton : FB_BannerPalmButton;
	topCoverLiftedFault : FB_Fault(name := 'Top Cover Lifeted During Cycle');
	amazonBPM : FB_AmazonThroughput();
	printerLabel : FB_PrinterSerial();
	autoModeTimer : Standard.TON;
	autoModeKeepCycling : BOOL;
	autoModeInitiateCycleONS : FB_ONS;
	cycleComplete : FB_ONS;
	hIecTask : RTS_IEC_HANDLE;//Declaration of the variable hIecTask
	teachPhotoeyeTimer : Standard.TOF() := (PT := T#3S);
	//variables for the state timer
	stateTimer:TON;
	laststate: INT;
	count_index :INT :=0;
	clr:BOOL:=FALSE;
	speedTracking : ARRAY[0..20] OF ARRAY[0..20] OF TIME;
	speedTracking_mt : ARRAY[0..20] OF ARRAY[0..20] OF TIME:=[21([21(T#0S)])];
	state_index : INT:=0;
	hold: BOOL;
	loadPlateInterlocks: DINT := 0;
	resetHold: Ton;
END_VAR(*#-#-#-#-#-#-#-#-#-#---Implementation---#-#-#-#-#-#-#-#-#-#-#-#-#*)

//	Program: PLC_PRG
//	Description: Base program for the 1179/1181 SX.
//
//	Created by: Ben Hess
//	Created Date:

IO_Map();
// Initialze global objects on first scan
IF NOT firstScanDone THEN
	GlobalObjects.CollectionOfInitialzable.InitializeAll();
	GlobalObjects.CollectionOfLoggable.RegisterAll(internalLogger := Globals.SystemLog);
	GlobalObjects.CollectionOfFaults.FaultUpdateForHMI();
	hIecTask := IecTaskGetCurrent(0);
	IecTaskDisableWatchdog(hIecTask); // Watchdog disabled
	firstScanDone := TRUE;
END_IF
IF firstAborted AND UN00_SXMachine.currentState = PACK_ML.State.Aborted THEN
	firstAborted := FALSE;
END_IF
// Use fault collection for faultActive indication
HMIData.faultActive := GlobalObjects.CollectionOfActiveFaults.faultActive;

// Cycle start conditions
// Auto mode dwell timer
autoModeTimer(PT := TO_TIME(HMIData.autoModeDwell * 1000), IN := autoModeKeepCycling AND UN00_SXMachine.currentState = PACK_ML.State.Execute AND NOT HMIData.inCycle);
// Start from Cycle Start input
cycleStartONS(clk := iCycleStart);
// All start conditions
IF HMIData.initiateCycle OR cycleStartONS.OSR OR autoModeTimer.Q THEN
	IF UN00_SXMachine.currentState = PACK_ML.State.Execute AND NOT HMIData.inCycle THEN
		EM01_SXBaggerHead.StartCycle();
		IF HMIData.autoModeEnable THEN
			autoModeKeepCycling := TRUE;
		END_IF
	END_IF
	HMIData.initiateCycle := FALSE;
END_IF
// Unlatch flag for auto mode when faulted or stopped
IF UN00_SXMachine.currentState <> PACK_ML.State.Execute OR HMIData.ackAllFaults OR NOT HMIData.autoModeEnable THEN
	autoModeKeepCycling := FALSE;
END_IF

// Only faults execute automatically to handle acking and clearing without being run in each FB that contains them
IF firstScanDone THEN
	GlobalObjects.CollectionOfExecutable.ExecuteAll();
END_IF

// Barcode Verifier manual trigger
IF HMIData.barcodeVerifierTrigger THEN
	baggerCM.barcodeVerifier.TriggerImmediate();
	HMIData.barcodeVerifierTrigger := FALSE;
END_IF

// Printer sample label sending
IF HMIData.sendSampleLabels AND NOT printerLabel.xExecute THEN
	printerLabel.xExecute := TRUE;
	printerLabel.sendSampleLabel := TRUE;
	printerLabel.sendClearLabel := FALSE;
	HMIData.sendSampleLabels := FALSE;
ELSIF HMIData.clearAllLabels AND NOT printerLabel.xExecute THEN
	printerLabel.xExecute := TRUE;
	printerLabel.sendSampleLabel := FALSE;
	printerLabel.sendClearLabel := TRUE;
	HMIData.clearAllLabels := FALSE;
END_IF

IF printerLabel.xDone THEN
	printerLabel.xExecute := FALSE;
END_IF
printerLabel();

// Run collection of bagger control modules
baggerCM(inhibitMotion:= firstAborted);
dischargeCM(loadPlateInterlocks:= loadPlateInterlocks);

// Set bagger head control modules
EM01_SXBaggerHead(
	bagOpenFingers:= baggerCM.dummyBOF,
	sealFlatteners:= baggerCM.dummySealFlatteners,
	sealer:= baggerCM.sealWire,
	pressureBar:= baggerCM.dualMotorPassthrough,
	printer:= baggerCM.labelPrinter,
	bagDelivery:= baggercm.bagDelivery,
	vacuumBagOpen:= baggerCM.dummyVacuumCups,
	IBD:= baggerCM.IBD,
	loadPlate:= dischargeCM.loadPlate,
	barcodeVerifier:= baggerCM.barcodeVerifier,
	bagOpenAssistEnabled:= FALSE,
	bagOpenSensorEnabled:= FALSE,
	cancelPrint := HMIData.printerCancelRequest,
	separateBeforeSealEnabled:= HMIData.separateBeforeSeal,
	bagOpenRetrySetting:= ,
	newJobLoaded:= ,
	vacuumDwell:= ,
	bagOpenRetryCount=> ,
	failedToOpenBag=> );

EM02_SXDischarge();

// Machine unit
UN00_SXMachine(faultActive:= HMIData.faultActive, resetMachine := HMIData.ackAllFaults, homeMachine := HMIData.homeMachine, currentState=> , baggerHead:= EM01_SXBaggerHead, discharge:= EM02_SXDischarge);

// Trigger fault if top cover lifted during cycle
IF HMIData.inCycle AND NOT iTopCoverClosed THEN
	topCoverLiftedFault.Trigger();
END_IF

// Banner palm button has 4 states - off, solid green, 50/50 green/white rotating, and flashing red
palmButton(
	baggerReady:= UN00_SXMachine.currentState = PACK_ML.State.Execute,
	baggerFaulted:= HMIData.faultActive,
	baggerInCycle:= HMIData.inCycle,
	palmState0Output=> oPalmButton0,
	palmState1Output=> oPalmButton1);

//
// HMI Mapping
//
//code to add timer to track duration in states
stateTimer(PT:=T#10000S);
stateTimer.IN := UN00_SXMachine.baggerManager.BaggerAutoMode.baggerCycleActive;
IF clr THEN
	speedTracking:=speedTracking_mt;
	clr:=FALSE;
END_IF
IF UN00_SXMachine.baggerManager.BaggerAutoMode.baggerCycleActive AND NOT hold THEN
		count_index := count_index +1;
		hold:=TRUE;
ELSIF hold AND NOT UN00_SXMachine.baggerManager.BaggerAutoMode.baggerCycleActive THEN
	hold := FALSE;
END_IF
IF stateTimer.ET>T#0MS THEN
	speedTracking[state_index][count_index] := stateTimer.ET;
END_IF
IF count_index >=20 THEN
	count_index :=0;
END_IF
resetHold(IN:=HMIData.ackAllFaults,PT:=T#100MS);
IF HMIData.ackAllFaults THEN
	IF UN00_SXMachine.currentState = PACK_ML.State.Resetting OR resetHold.Q THEN
		HMIData.ackAllFaults:= FALSE;
	END_IF
END_IF
//End modded code
// Send the list of active fault strings to HMI for viewing
HMIData.activeFaults := GlobalObjects.CollectionOfActiveFaults.ObjNames;
hmiFaultMessage(faultActive:= GlobalObjects.CollectionOfActiveFaults.faultActive,faultList:= GlobalObjects.CollectionOfActiveFaults.ObjNames);
HMIData.faultMessage:=hmiFaultMessage.faultMessagestr;
HMIData.inCycle := UN00_SXMachine.baggerManager.BaggerAutoMode.baggerCycleActive;
// PackML state to string for HMI
HMIData.currentPackMLState := UN00_SXMachine.baggerManager.BaggerAutoMode.currentBaggerState;

oFansEnable := NOT HMIData.standbyActive;

// Banner manager takes care of the Multistate lamp used as a banner on the proface
bannerManager(
	baggerNotReady:= NOT UN00_SXMachine.currentState = PACK_ML.State.Execute,
	baggerReady:= UN00_SXMachine.currentState = PACK_ML.State.Execute AND NOT HMIData.inCycle,
	baggerInCycle:= HMIData.inCycle,
	noBagCoveringEye:= baggerCM.bagDelivery.noBagOverEye.Active,
	bagFailedToSeperate:= baggerCM.bagDelivery.bagFailedToSeparate.Active,
	pbarObstruction:= baggerCM.dualMotorPassthrough.pressureBarObstructed.Active,
	lightCurtainViolation:= ,
	printHeadFTR:= baggerCM.labelPrinter.printHeadFailToRaise.Active,
	printHeadFTL:= baggerCM.labelPrinter.printHeadFailToLower.Active,
	barcodeFault:= EM01_SXBaggerHead.barcodeVerificationFailed.Active,
	tooManyPartsCounted:= ,
	jawFailedToClose:= baggerCM.dualMotorPassthrough.failedToClose.Active,
	jawFailedToHome:= baggerCM.dualMotorPassthrough.failedToHome.Active,
	filmFeedMotorFault:=  baggerCM.bagDeliveryFrontMotor.error OR baggerCM.bagDelivery.reverseFault.Active,
	jawMotionFault:= baggerCM.jawFrontMotor.error OR baggerCM.dualMotorPassthrough.frontMotorFault.Active OR baggerCM.dualMotorPassthrough.frontMotorCommFault.Active,
	//jawMotionFault:= baggerCM.dualMotorPassthrough.bothMotorsFault.Active,
	waitingOnPrinter:= UN00_SXMachine.baggerManager.BaggerAutoMode.releaseAndFeedSubState = RELEASE_FEED_STATES.WaitForPrinter,
	waitingOnFiller:= ,
	batchCounterDone:= ,
	jawNotHomed:= NOT baggerCM.dualMotorPassthrough.IsHomed AND NOT HMIData.inCycle,
	cycleBaggerTForFiller:= ,
	machineNotTested:=  HMIData.bagsMade < 1000,
	//loadPlateMotorNotHomed:= NOT baggerCM.loadPlate.IsHomed AND baggerCM.loadPlate.OptionActive,
	//loadPlateMotorFaulted:= baggerCM.loadPlate.motorFault.Active,
	//loadPlateMotorCommF:= baggerCM.loadPlate.motorCommFault.Active,
	topCoverLiftedFault:= topCoverLiftedFault.Active,
	topCoverLiftedWarning:= NOT iTopCoverClosed AND NOT HMIData.inCycle,
	//IBDMotorNotHomed:= NOT baggerCM.IBD.IsHomed AND baggerCM.IBD.OptionActive AND NOT HMIData.inCycle,
	//IBDMotorFaulted:= baggerCM.IBD.IBDMotorFault.Active,
	//IBDMotorCommF:= baggerCM.IBD.IBDMotorCommFault.Active,
	printerRibbonFault := baggerCM.labelPrinter.ribbonFault.Active,
	printerServiceRequired := baggerCM.labelPrinter.serviceRequired.Active,
	jawFailedToOpen:= baggerCM.dualMotorPassthrough.failedToOpen.Active,
	IBDFailedToClose:= baggerCM.dualMotorPassthrough.failedToClose.Active,
	//IBDFailedToOpen:= baggerCM.IBD.failedToOpen.Active,
	messageDisplayIndication=> HMIData.bannerMessageIndication);

// Ready indications for bagger control modules
HMIData.printerReady := baggerCM.labelPrinter.Ready;
HMIData.bagDeliveryReady := baggerCM.bagDelivery.Ready;
//HMIData.loadPlateReady := baggerCM.loadPlate.Ready;
HMIData.jawReady := baggerCM.dualMotorPassthrough.Ready;
HMIData.bcvReady := baggerCM.barcodeVerifier.Ready;
HMIData.IBDReady := baggerCM.IBD.Ready;

// Motor data to HMI for troubleshooting
HMIData.frontJawMotorData.ActPos := baggerCM.jawFrontMotor.ActPos;
HMIData.frontJawMotorData.CommandedPos := baggerCM.jawFrontMotor.TargetPosDist;
HMIData.frontJawMotorData.CurrentAlarmCode := baggerCM.jawFrontMotor.alarmCode;

//HMIData.bagDeliveryMotorData.alarmCode := baggerCM.bagDeliveryFrontMotor.alarmCode;;

// Cycle time and bags made counters
HMIData.cycleTime := UN00_SXMachine.baggerManager.BaggerAutoMode.cycleTime;
HMIData.inCycle := UN00_SXMachine.baggerManager.BaggerAutoMode.cycleTimer.IN;
cycleComplete(CLK := UN00_SXMachine.baggerManager.BaggerAutoMode.cycleComplete);
IF cycleComplete.OSR THEN
	HMIData.bagsMade := HMIData.bagsMade + 1;
END_IF

// Printer and Barcode Verifier combination enable/disable
HMIData.printerAndVerifierEnableIndication := HMIData.printerInUse AND HMIData.barcodeVerifierInUse;
IF HMIData.printerAndVerifierEnablePB THEN
	IF HMIData.printerAndVerifierEnableIndication THEN
		HMIData.printerInUse := FALSE;
		HMIData.barcodeVerifierInUse := FALSE;
	ELSE
		HMIData.printerInstalled := TRUE;
		HMIData.barcodeVerifierInstalled := TRUE;
		HMIData.printerInUse := TRUE;
		HMIData.barcodeVerifierInUse := TRUE;
	END_IF
	HMIData.printerAndVerifierEnablePB := FALSE;
END_IF

// Position Indications for service commands
HMIData.jawService.extendedFeedback := baggerCM.dualMotorPassthrough.IsFullyOpen;
HMIData.jawService.retractedFeedback := baggerCM.dualMotorPassthrough.IsFullyClosed;

//HMIData.IBDService.extendedFeedback := baggerCM.IBD._isFullyOpen;
//HMIData.IBDService.retractedFeedback := NOT baggerCM.IBD._isFullyOpen;

HMIData.printHeadService.extendedFeedback := oLowerPrinthead;
HMIData.printHeadService.retractedFeedback := NOT oLowerPrinthead;

// Amazon Bags per minute throughput calculator
amazonBPM(
	inCycle:= HMIData.inCycle,
	runtimeTimeout:= ,
	reset:= HMIData.BPMReset,
	BPM=> HMIData.BPMBagsPerMinute,
	BPMCycles=> HMIData.BPMBagsMade,
	BPMSeconds=> ,
	BPMIndication=> HMIData.BPMActiveTime);
